(* Logix 5000 project; controller Factory_io vendor 1 type 14 code 15 rev 16.42; software revision 16.03 *)

TASK MainTask (continuous, watchdog 500 ms) : MainProgram

MODULES
   Local : vendor 1 type 14 code 15 (SoftLogixController 2, rev 16.42)
END_MODULES

ADD_ON_INSTRUCTION Add_On_Pusher   (* revision 1.0 *)
VAR_INPUT
   Modo_Op : BOOL; {visible}   // Auto 0 Manual 1
END_VAR
VAR_OUTPUT
   AutoRunning : BOOL;   // Pusher en auto
   ManuRunnig : BOOL;   // Pusher en manual
END_VAR
VAR_INPUT
   cmdRun : BOOL; {visible}   // Activar Pusher Automatico
   cmdStop : BOOL;   // Parada Auto Pusher
END_VAR
VAR_OUTPUT
   StsRunning : BOOL; {visible}   // Salida fisica del PLC
END_VAR
VAR_INPUT
   HMI_Run : BOOL; {visible}   // Pusher Manual
   sensorBackL : BOOL;   // Sensor de posicion del basculante
   sensorFront : BOOL;   // Sensor Posicion basculante
END_VAR
VAR
   HMI_Stop : BOOL;
   expandir : BOOL;
   Encoger : BOOL;   // Accion cuando el sensor Back esta en 0
END_VAR

ROUTINE Logic   (* ladder *)
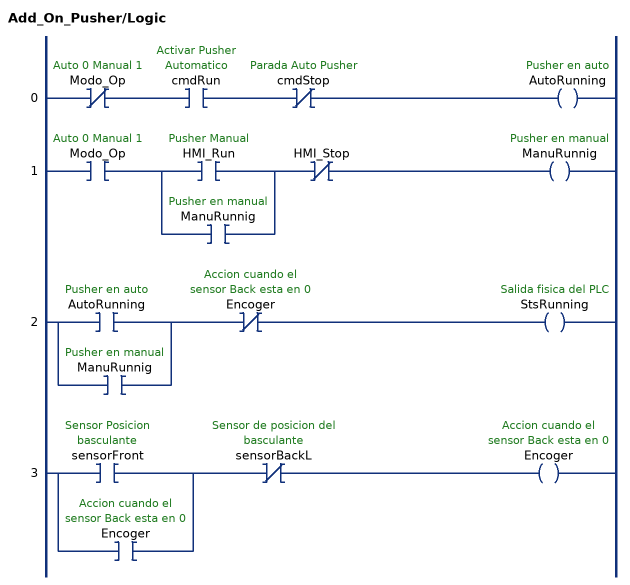
   0: XIO(Modo_Op)XIC(cmdRun)XIO(cmdStop)OTE(AutoRunning);
   1: XIC(Modo_Op)[XIC(HMI_Run) ,XIC(ManuRunnig) ]XIO(HMI_Stop)OTE(ManuRunnig);
   2: [XIC(AutoRunning) ,XIC(ManuRunnig) ]XIO(Encoger)OTE(StsRunning);
   3: [XIC(sensorFront) ,XIC(Encoger) ]XIO(sensorBackL)OTE(Encoger);
END_ROUTINE
END_ADD_ON_INSTRUCTION

ADD_ON_INSTRUCTION Bascula   (* revision 1.0 *)
VAR
   Modo_Op : BOOL;
   HMI_Run : BOOL;
   HMI_Stop : BOOL;
   ManuRunnig : BOOL;
   cmdRun : BOOL;
   cmdStop : BOOL;
   AutoRunning : BOOL;
   Bascula_On : BOOL;
   Peso : REAL;
   Direccion_Derecha : BOOL;
   Ruedas : BOOL;
   Direccion_Izquierda : BOOL;
   Pieza_Izquierda : BOOL;
   Pieza_Derecha : BOOL;
   Sensor_Out_Izquierda : BOOL;
   Sensor_Out_Derecha : BOOL;
END_VAR

ROUTINE Logic   (* ladder *)
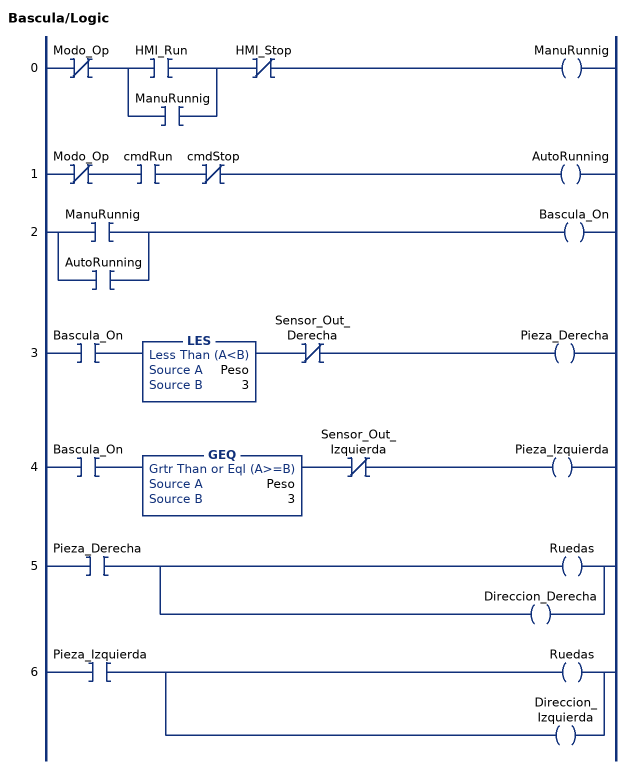
   0: XIO(Modo_Op)[XIC(HMI_Run) ,XIC(ManuRunnig) ]XIO(HMI_Stop)OTE(ManuRunnig);
   1: XIO(Modo_Op)XIC(cmdRun)XIO(cmdStop)OTE(AutoRunning);
   2: [XIC(ManuRunnig) ,XIC(AutoRunning) ]OTE(Bascula_On);
   3: XIC(Bascula_On)LES(Peso,3)XIO(Sensor_Out_Derecha)OTE(Pieza_Derecha);
   4: XIC(Bascula_On)GEQ(Peso,3)XIO(Sensor_Out_Izquierda)OTE(Pieza_Izquierda);
   5: XIC(Pieza_Derecha)[OTE(Ruedas) ,OTE(Direccion_Derecha) ];
   6: XIC(Pieza_Izquierda)[OTE(Ruedas) ,OTE(Direccion_Izquierda) ];
END_ROUTINE
END_ADD_ON_INSTRUCTION

ADD_ON_INSTRUCTION Brazos_Roboticos   (* revision 1.0 *)
VAR_INPUT
   Modo_Op : BOOL; {visible}   // Auto 0 Manual 1
   CmdStop : BOOL; {visible}   // Para desactivar el brazo en modo auto
   CmdRun : BOOL; {visible}   // Para activar el brazo en modo auto
   HMI_Run : BOOL; {visible}   // Para activar el brazo en modo manual
   HMI_Stop : BOOL; {visible}   // Para desactivar el brazo en modo manual
END_VAR
VAR_OUTPUT
   autoRunning : BOOL;   // brazo funcionando en modo auto
   manRunning : BOOL;   // brazo funcionando en modo manual
   StsRunning : BOOL; {visible}   // salida fisica al PLC
END_VAR
VAR_INPUT
   InpRunning : BOOL; {visible}   // Deteccion de falla en el equipo
END_VAR
VAR_OUTPUT
   StsFallo : BOOL; {visible}   // Refleja falla del equipo
   StsStop : BOOL;
END_VAR
VAR
   Timer_TT : BOOL;
   Timer_RES : BOOL;
   Timer_EN : BOOL;
   Timer_DN : BOOL;
   RTO : TIMER;
END_VAR

ROUTINE Logic   (* ladder *)
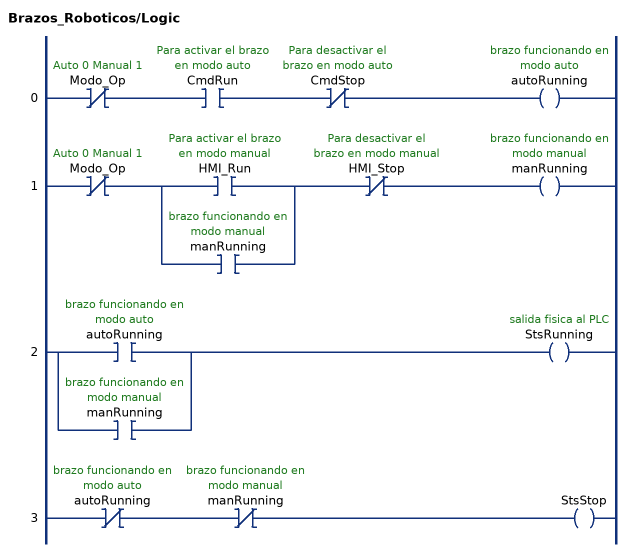
   0: XIO(Modo_Op)XIC(CmdRun)XIO(CmdStop)OTE(autoRunning);
   1: XIO(Modo_Op)[XIC(HMI_Run) ,XIC(manRunning) ]XIO(HMI_Stop)OTE(manRunning);
   2: [XIC(autoRunning) ,XIC(manRunning) ]OTE(StsRunning);
   3: XIO(autoRunning)XIO(manRunning)OTE(StsStop);
END_ROUTINE
END_ADD_ON_INSTRUCTION

ADD_ON_INSTRUCTION Motores   (* revision 1.0 *)
VAR_INPUT
   MODO_OPERACION : BOOL; {visible}
   Cmd_Start : BOOL; {visible}   // Comando para activar el motor en modo auto
   Cmd_Stop : BOOL; {visible}   // Comando para detener el motor en auto
   HMI_Run : BOOL;   // Comando para activar el motor en manual
   HMI_Stop : BOOL;   // Comando para detener el motor en manual
   Inp_Running : BOOL; {visible}   // Confirmacion de arranque del motor
END_VAR
VAR_OUTPUT
   Sts_Running : BOOL; {visible}   // Estado de arranque del motor
   Sts_Running_Pass : BOOL; {visible}   // Estado de motor en la falla
END_VAR
VAR
   Timer_Pass : TIMER := (PRE := 5000);
   Manu_Running : BOOL;
   Auto_Running : BOOL;
END_VAR

ROUTINE Logic   (* ladder *)
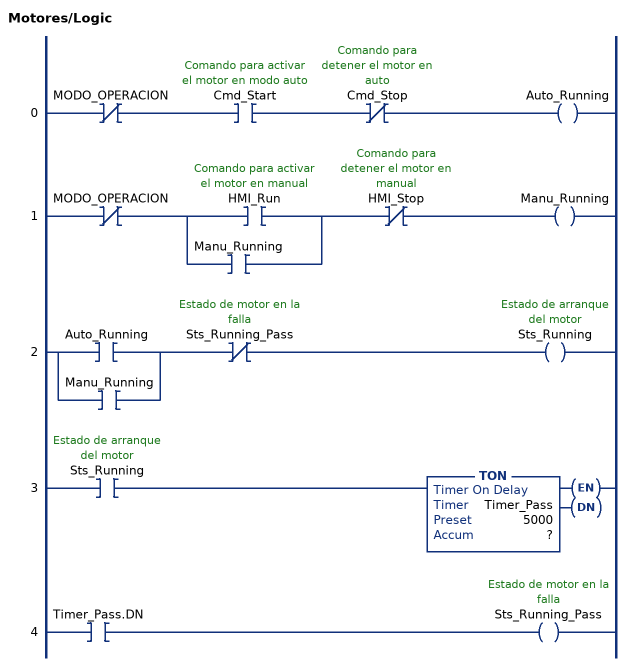
   0: XIO(MODO_OPERACION)XIC(Cmd_Start)XIO(Cmd_Stop)OTE(Auto_Running);
   1: XIO(MODO_OPERACION)[XIC(HMI_Run) ,XIC(Manu_Running) ]XIO(HMI_Stop)OTE(Manu_Running);
   2: [XIC(Auto_Running) ,XIC(Manu_Running) ]XIO(Sts_Running_Pass)OTE(Sts_Running);
   3: XIC(Sts_Running)TON(Timer_Pass,?,?);
   4: XIC(Timer_Pass.DN)OTE(Sts_Running_Pass);
END_ROUTINE
END_ADD_ON_INSTRUCTION

ADD_ON_INSTRUCTION Pick_xyz_avanzado   (* revision 1.0 *)
VAR_INPUT
   Modo_Op : BOOL; {visible}   // Auto 0 Manual 1
END_VAR
VAR_OUTPUT
   AutoRunning : BOOL;   // brazo en auto
   ManuRunnig : BOOL;   // Brazo en manual
END_VAR
VAR_INPUT
   cmdRun : BOOL; {visible}   // Activar Brazo Automatico
   cmdStop : BOOL;   // Parada Auto brazo
END_VAR
VAR_OUTPUT
   StsRunning : BOOL; {visible}   // Salida fisica del PLC
END_VAR
VAR_INPUT
   HMI_Run : BOOL; {visible}   // Brazo Manual
END_VAR
VAR
   HMI_Stop : BOOL;
   maquina_Operando : BOOL;
   Posicion_X : DINT;
   Posicion_Y : DINT;
   Posicion_Z : DINT;
   Etapa_Agarrar : BOOL;
   Etapa_Soltar_1 : BOOL;
   Etapa_Soltar_2 : BOOL;
   Etapa_Soltar_3 : BOOL;
END_VAR

ROUTINE Logic   (* ladder *)
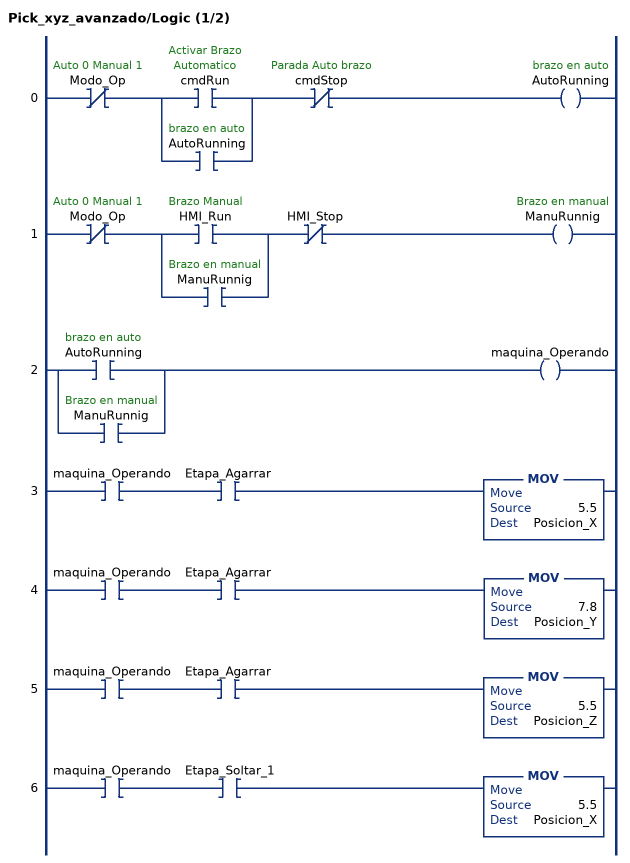
   0: XIO(Modo_Op)[XIC(cmdRun) ,XIC(AutoRunning) ]XIO(cmdStop)OTE(AutoRunning);
   1: XIO(Modo_Op)[XIC(HMI_Run) ,XIC(ManuRunnig) ]XIO(HMI_Stop)OTE(ManuRunnig);
   2: [XIC(AutoRunning) ,XIC(ManuRunnig) ]OTE(maquina_Operando);
   3: XIC(maquina_Operando)XIC(Etapa_Agarrar)MOV(5.5,Posicion_X);
   4: XIC(maquina_Operando)XIC(Etapa_Agarrar)MOV(7.8,Posicion_Y);
   5: XIC(maquina_Operando)XIC(Etapa_Agarrar)MOV(5.5,Posicion_Z);
   6: XIC(maquina_Operando)XIC(Etapa_Soltar_1)MOV(5.5,Posicion_X);
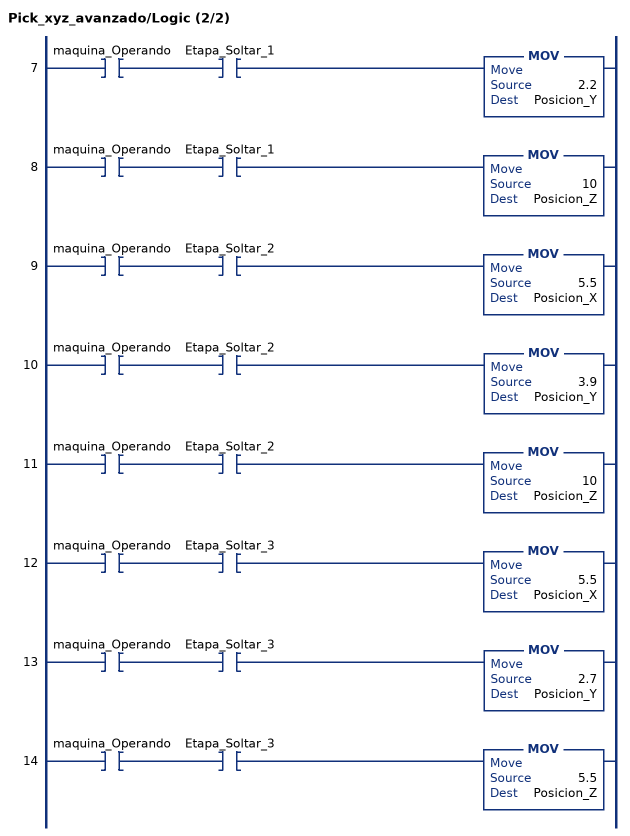
   7: XIC(maquina_Operando)XIC(Etapa_Soltar_1)MOV(2.2,Posicion_Y);
   8: XIC(maquina_Operando)XIC(Etapa_Soltar_1)MOV(10,Posicion_Z);
   9: XIC(maquina_Operando)XIC(Etapa_Soltar_2)MOV(5.5,Posicion_X);
   10: XIC(maquina_Operando)XIC(Etapa_Soltar_2)MOV(3.9,Posicion_Y);
   11: XIC(maquina_Operando)XIC(Etapa_Soltar_2)MOV(10,Posicion_Z);
   12: XIC(maquina_Operando)XIC(Etapa_Soltar_3)MOV(5.5,Posicion_X);
   13: XIC(maquina_Operando)XIC(Etapa_Soltar_3)MOV(2.7,Posicion_Y);
   14: XIC(maquina_Operando)XIC(Etapa_Soltar_3)MOV(5.5,Posicion_Z);
END_ROUTINE
END_ADD_ON_INSTRUCTION

VAR_GLOBAL   (* controller tags *)
   Add_ON_BrazosRoboticos_1 : Brazos_Roboticos;
   Add_ON_BrazosRoboticos_2 : Brazos_Roboticos;
   Add_Pusher_01 : Add_On_Pusher;
   Add_Pusher_02 : Add_On_Pusher;
   Add_Pusher_03 : Add_On_Pusher;
   Agarrar_Soltar : BOOL;
   BOOL_IN_0 : ALIAS FOR Sensor_In1_verde;
   BOOL_IN_1 : ALIAS FOR Sensor_In2_verde;
   BOOL_IN_10 : ALIAS FOR Add_Pusher_03.sensorFront;
   BOOL_IN_11 : ALIAS FOR Add_Pusher_01.sensorBackL;
   BOOL_IN_12 : ALIAS FOR Add_Pusher_02.sensorBackL;
   BOOL_IN_13 : ALIAS FOR Add_Pusher_03.sensorBackL;
   BOOL_IN_14 : ALIAS FOR Difuse_Sensor_In;
   BOOL_IN_15 : ALIAS FOR Difuse_Sensor_Out;
   BOOL_IN_16 : ALIAS FOR Pieza_In;
   BOOL_IN_17 : ALIAS FOR sensor_In_Peso;
   BOOL_IN_18 : ALIAS FOR sensor_Out_banda_der;
   BOOL_IN_19 : ALIAS FOR sensor_Out_banda_Izq;
   BOOL_IN_2 : ALIAS FOR Sensor_Out1;
   BOOL_IN_20 : ALIAS FOR Parada_Peso;
   BOOL_IN_21 : ALIAS FOR Modo_Operacion;
   BOOL_IN_22 : ALIAS FOR STOP;
   BOOL_IN_3 : ALIAS FOR Sensor_Out2;
   BOOL_IN_4 : ALIAS FOR START;
   BOOL_IN_5 : ALIAS FOR sensorVerde;
   BOOL_IN_6 : ALIAS FOR sensorAzul;
   BOOL_IN_7 : ALIAS FOR sensorGris;
   BOOL_IN_8 : ALIAS FOR Add_Pusher_01.sensorFront;
   BOOL_IN_9 : ALIAS FOR Add_Pusher_02.sensorFront;
   BOOL_OUT_0 : ALIAS FOR cintaEntrada1.Sts_Running;
   BOOL_OUT_1 : ALIAS FOR cintaEntrada2.Sts_Running;
   BOOL_OUT_10 : ALIAS FOR cintaEntradaPush2.Sts_Running;
   BOOL_OUT_11 : ALIAS FOR Add_Pusher_01.StsRunning;
   BOOL_OUT_12 : ALIAS FOR Add_Pusher_02.StsRunning;
   BOOL_OUT_13 : ALIAS FOR Add_Pusher_03.StsRunning;
   BOOL_OUT_14 : ALIAS FOR Subir_Bajar;
   BOOL_OUT_15 : ALIAS FOR Agarrar_Soltar;
   BOOL_OUT_16 : ALIAS FOR Pasa_Banda;
   BOOL_OUT_17 : ALIAS FOR Cinta_In_Pick1.Sts_Running;
   BOOL_OUT_18 : ALIAS FOR Cinta_In_Pick2.Sts_Running;
   BOOL_OUT_19 : ALIAS FOR Cinta_In_Pick3.Sts_Running;
   BOOL_OUT_2 : ALIAS FOR cintaSalida_01.Sts_Running;
   BOOL_OUT_20 : ALIAS FOR Cinta_In_Pick4.Sts_Running;
   BOOL_OUT_21 : ALIAS FOR Cinta_In_Pick5.Sts_Running;
   BOOL_OUT_22 : ALIAS FOR Cinta_In_Pick6.Sts_Running;
   BOOL_OUT_23 : ALIAS FOR cintaPP.Sts_Running;
   BOOL_OUT_24 : ALIAS FOR movScale.Sts_Running;
   BOOL_OUT_25 : ALIAS FOR clasificaPlus.Sts_Running;
   BOOL_OUT_26 : ALIAS FOR clasificaDerecha.Sts_Running;
   BOOL_OUT_27 : ALIAS FOR clasificaIzq.Sts_Running;
   BOOL_OUT_28 : ALIAS FOR cintaPesoDer.Sts_Running;
   BOOL_OUT_29 : ALIAS FOR cintaPesoIzq.Sts_Running;
   BOOL_OUT_3 : ALIAS FOR cintaSalida_02.Sts_Running;
   BOOL_OUT_30 : ALIAS FOR Luz_Verde;
   BOOL_OUT_31 : ALIAS FOR Luz_stop;
   BOOL_OUT_4 : ALIAS FOR Maquina_1;
   BOOL_OUT_5 : ALIAS FOR Maquina_2;
   BOOL_OUT_6 : ALIAS FOR cintaRecorrido1.Sts_Running;
   BOOL_OUT_7 : ALIAS FOR cintaRecorrido2.Sts_Running;
   BOOL_OUT_8 : ALIAS FOR cintarecorrido3.Sts_Running;
   BOOL_OUT_9 : ALIAS FOR cintaEntradaPush1.Sts_Running;
   cinta : Motores;
   Cinta_In_Pick1 : Motores;
   Cinta_In_Pick2 : Motores;
   Cinta_In_Pick3 : Motores;
   Cinta_In_Pick4 : Motores;
   Cinta_In_Pick5 : Motores;
   Cinta_In_Pick6 : Motores;
   cintaEntrada1 : Motores;
   cintaEntrada1_01 : Motores;
   cintaEntrada1_02 : Motores;
   cintaEntrada2 : Motores;
   cintaEntradaPush1 : Motores;
   cintaEntradaPush2 : Motores;
   cintaPeso : Motores;
   cintaPesoDer : Motores;
   cintaPesoIzq : Motores;
   cintaPP : Motores;
   cintaRecorrido1 : Motores;
   cintaRecorrido2 : Motores;
   cintarecorrido3 : Motores;
   cintarecorrido3_01 : Motores;
   cintaSalida_01 : Motores;
   cintaSalida_02 : Motores;
   cintaSalida_03 : Motores;
   cintaSalida_04 : Motores;
   cintaSalida_05 : Motores;
   cintaSalida_06 : Motores;
   clasificaDerecha : Motores;
   clasificaIzq : Motores;
   clasificaPlus : Motores;
   Difuse_Sensor_In : BOOL;
   Difuse_Sensor_Out : BOOL;
   FLOAT_IN_0 : ALIAS FOR SensorPeso;
   INICO_001 : SFC_STEP := (Status := 16#0800_0201, DN := 1, T := 16, TMax := 20306, Count := 4);
   INICO_002 : SFC_STEP := (Status := 16#0800_0201, DN := 1, T := 16, TMax := 20306, Count := 4);
   Luz_stop : BOOL;
   Luz_Verde : BOOL;
   Maquina_1 : BOOL;
   Maquina_2 : BOOL;
   Modo_Operacion : BOOL;   // 0 AUTO 1 MANUAL
   movScale : Motores;
   Parada_Peso : BOOL;
   Pasa_Banda : BOOL;
   Pick_On : BOOL;
   Pieza_In : BOOL;
   Sensor_In1_verde : BOOL := 1;
   Sensor_In2_verde : BOOL := 1;
   sensor_In_Peso : BOOL;
   Sensor_Out1 : BOOL := 1;
   Sensor_Out2 : BOOL := 1;
   sensor_Out_banda_der : BOOL;
   sensor_Out_banda_Izq : BOOL;
   sensorAzul : BOOL;
   sensorGris : BOOL;
   SensorPeso : REAL;
   sensorVerde : BOOL;
   START : BOOL;
   STOP : BOOL;
   Subir_Bajar : BOOL;
   SYS_ON : BOOL;
END_VAR

PROGRAM MainProgram   (* main routine MainRoutine *)
VAR
   Action_000 : SFC_ACTION := (Status := 16#c000_0000, A := 1, Q := 1, Count := 4);
   Action_001 : SFC_ACTION := (Count := 4);
   Action_002 : SFC_ACTION := (Count := 4);
   Action_003 : SFC_ACTION := (Count := 3);
   Action_004 : SFC_ACTION := (Count := 4);
   Action_005 : SFC_ACTION := (Status := 16#c000_0000, A := 1, Q := 1, Count := 4);
   Action_006 : SFC_ACTION := (Count := 3);
   Action_007 : SFC_ACTION := (Count := 4);
   Action_008 : SFC_ACTION;
   Action_009 : SFC_ACTION;
   Action_010 : SFC_ACTION;
   Action_011 : SFC_ACTION;
   Action_012 : SFC_ACTION;
   Action_013 : SFC_ACTION;
   Action_014 : SFC_ACTION;
   Action_015 : SFC_ACTION;
   Action_016 : SFC_ACTION;
   Action_017 : SFC_ACTION;
   Action_018 : SFC_ACTION;
   Action_019 : SFC_ACTION;
   Motores_01 : Motores := (Cmd_Start := 1);
   Motores_02 : Motores := (Cmd_Start := 1);
   Motores_03 : Motores := (Cmd_Start := 1);
   Motores_04 : Motores := (Cmd_Start := 1);
   Step_000 : SFC_STEP;
   Step_001 : SFC_STEP;
   Step_002 : SFC_STEP := (Status := 16#0800_0001, DN := 1, PRE := 400, T := 314, TMax := 327, Count := 4);
   Step_003 : SFC_STEP := (Status := 16#0800_0001, DN := 1, T := 2150, TMax := 2212, Count := 4);
   Step_004 : SFC_STEP := (Status := 16#0800_0001, DN := 1, T := 2192, TMax := 2234, Count := 4);
   Step_005 : SFC_STEP := (PRE := 300);
   Step_006 : SFC_STEP := (Status := 16#0800_0001, DN := 1, T := 18, TMax := 19, Count := 4);
   Step_007 : SFC_STEP := (Status := 16#0800_0001, DN := 1, T := 18, TMax := 19, Count := 4);
   Step_008 : SFC_STEP := (Status := 16#a800_0001, X := 1, SA := 1, DN := 1, T := 60168, TMax := 60168, Count := 4);
   Step_009 : SFC_STEP := (Status := 16#0800_0001, DN := 1, PRE := 6000, T := 5019, TMax := 5019, Count := 3);
   Step_010 : SFC_STEP := (Status := 16#a800_0001, X := 1, SA := 1, DN := 1, T := 60169, TMax := 60169, Count := 4);
   Step_011 : SFC_STEP := (Status := 16#0800_0001, DN := 1, PRE := 400, T := 314, TMax := 322, Count := 4);
   Step_012 : SFC_STEP := (Status := 16#0800_0001, DN := 1, PRE := 2000, T := 5019, TMax := 5019, Count := 3);
   Step_013 : SFC_STEP;
   Step_014 : SFC_STEP;
   Step_015 : SFC_STEP := (PRE := 300);
   Step_016 : SFC_STEP := (PRE := 400);
   Step_017 : SFC_STEP := (PRE := 400);
   Step_018 : SFC_STEP := (PRE := 1000);
   Step_019 : SFC_STEP;
   Step_020 : SFC_STEP := (PRE := 300);
   Step_021 : SFC_STEP := (PRE := 500);
   Step_022 : SFC_STEP := (PRE := 300);
   Step_023 : SFC_STEP;
   Step_024 : SFC_STEP;
   Step_025 : SFC_STEP := (PRE := 3100);
   Step_026 : SFC_STEP := (PRE := 3100);
   Step_027 : SFC_STEP;
   Step_028 : SFC_STEP := (PRE := 200);
   Tran_000 : BOOL;
   Tran_001 : BOOL := 1;
   Tran_002 : BOOL := 1;
   Tran_003 : BOOL := 1;
   Tran_004 : BOOL := 1;
   Tran_005 : BOOL := 1;
   Tran_006 : BOOL;
   Tran_007 : BOOL := 1;
   Tran_008 : BOOL := 1;
   Tran_009 : BOOL := 1;
   Tran_010 : BOOL := 1;
   Tran_011 : BOOL;
   Tran_012 : BOOL := 1;
   Tran_013 : BOOL;
   Tran_014 : BOOL;
   Tran_015 : BOOL;
   Tran_016 : BOOL;
   Tran_017 : BOOL;
   Tran_018 : BOOL;
   Tran_019 : BOOL;
   Tran_020 : BOOL;
   Tran_021 : BOOL;
   Tran_022 : BOOL;
   Tran_023 : BOOL;
   Tran_024 : BOOL;
   Tran_025 : BOOL;
   Tran_026 : BOOL;
   Tran_027 : BOOL;
   Tran_028 : BOOL;
END_VAR

ROUTINE BRAZOS_ROBOTICOS   (* sequential function chart *)
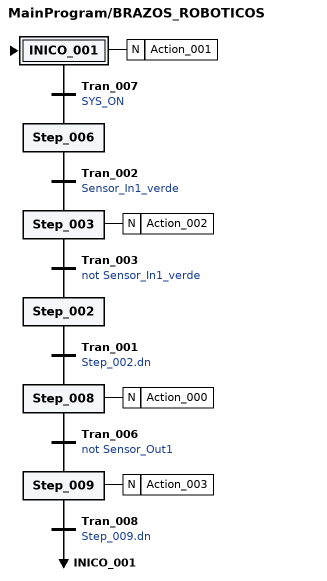
   INITIAL_STEP INICO_001:
      ACTION Action_001 (N):
         cintaEntrada1.Cmd_Start:=0;
         cintaSalida_01.Cmd_Start:=0;
         Maquina_1:=0;
         
         
         
      END_ACTION
   END_STEP
   TRANSITION Tran_007 FROM INICO_001 TO Step_006
      := SYS_ON
   END_TRANSITION
   STEP Step_006:
   END_STEP
   TRANSITION Tran_002 FROM Step_006 TO Step_003
      :=  Sensor_In1_verde
   END_TRANSITION
   STEP Step_003:
      ACTION Action_002 (N):
         cintaEntrada1.Cmd_Start:=1;
         
      END_ACTION
   END_STEP
   TRANSITION Tran_003 FROM Step_003 TO Step_002
      := not Sensor_In1_verde
   END_TRANSITION
   STEP Step_002:
   END_STEP
   TRANSITION Tran_001 FROM Step_002 TO Step_008
      := Step_002.dn
   END_TRANSITION
   STEP Step_008:
      ACTION Action_000 (N):
         cintaEntrada1.Cmd_Start:=0;
         Maquina_1:=1;
      END_ACTION
   END_STEP
   TRANSITION Tran_006 FROM Step_008 TO Step_009
      := not Sensor_Out1
   END_TRANSITION
   STEP Step_009:
      ACTION Action_003 (N):
         cintaSalida_01.Cmd_Start:=1;
         
         
      END_ACTION
   END_STEP
   TRANSITION Tran_008 FROM Step_009 TO INICO_001
      := Step_009.dn
   END_TRANSITION
END_ROUTINE

ROUTINE BRAZOS_ROBOTICOS_TAPAS   (* sequential function chart *)
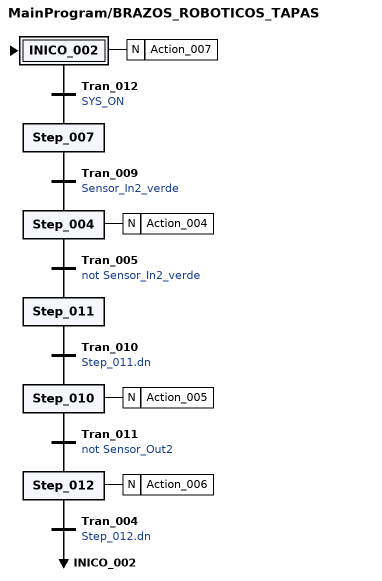
   INITIAL_STEP INICO_002:
      ACTION Action_007 (N):
         cintaEntrada2.Cmd_Start:=0;
         cintaSalida_02.Cmd_Start:=0;
         Maquina_2:=0;
         
         
         
      END_ACTION
   END_STEP
   TRANSITION Tran_012 FROM INICO_002 TO Step_007
      := SYS_ON
   END_TRANSITION
   STEP Step_007:
   END_STEP
   TRANSITION Tran_009 FROM Step_007 TO Step_004
      :=  Sensor_In2_verde
   END_TRANSITION
   STEP Step_004:
      ACTION Action_004 (N):
         cintaEntrada2.Cmd_Start:=1;
         
      END_ACTION
   END_STEP
   TRANSITION Tran_005 FROM Step_004 TO Step_011
      := not Sensor_In2_verde
   END_TRANSITION
   STEP Step_011:
   END_STEP
   TRANSITION Tran_010 FROM Step_011 TO Step_010
      := Step_011.dn
   END_TRANSITION
   STEP Step_010:
      ACTION Action_005 (N):
         cintaEntrada2.Cmd_Start:=0;
         Maquina_2:=1;
      END_ACTION
   END_STEP
   TRANSITION Tran_011 FROM Step_010 TO Step_012
      := not Sensor_Out2
   END_TRANSITION
   STEP Step_012:
      ACTION Action_006 (N):
         cintaSalida_02.Cmd_Start:=1;
         cintarecorrido3.Cmd_Start:=1;
         
         
      END_ACTION
   END_STEP
   TRANSITION Tran_004 FROM Step_012 TO INICO_002
      := Step_012.dn
   END_TRANSITION
END_ROUTINE

ROUTINE cintas_pushers   (* function block diagram *)
   SHEET 1
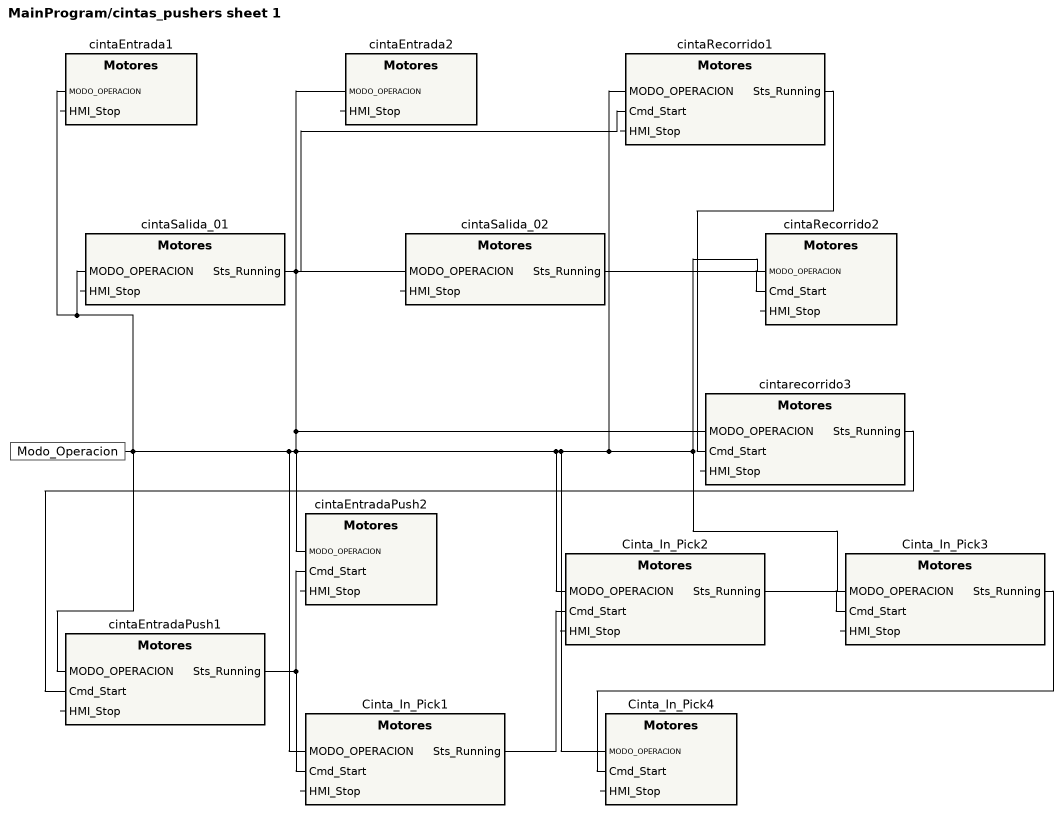
   cintaEntrada1 : Motores(MODO_OPERACION := Modo_Operacion);   // unwired pins: HMI_Stop
   cintaSalida_01 : Motores(MODO_OPERACION := Modo_Operacion);   // unwired pins: HMI_Stop
   cintaEntrada2 : Motores(MODO_OPERACION := Modo_Operacion);   // unwired pins: HMI_Stop
   cintaSalida_02 : Motores(MODO_OPERACION := Modo_Operacion);   // unwired pins: HMI_Stop
   cintaRecorrido1 : Motores(MODO_OPERACION := Modo_Operacion, Cmd_Start := cintaSalida_01.Sts_Running);   // unwired pins: HMI_Stop
   cintarecorrido3 : Motores(MODO_OPERACION := Modo_Operacion, Cmd_Start := cintaRecorrido1.Sts_Running);   // unwired pins: HMI_Stop
   cintaEntradaPush1 : Motores(MODO_OPERACION := Modo_Operacion, Cmd_Start := cintarecorrido3.Sts_Running);   // unwired pins: HMI_Stop
   cintaEntradaPush2 : Motores(MODO_OPERACION := Modo_Operacion, Cmd_Start := cintaEntradaPush1.Sts_Running);   // unwired pins: HMI_Stop
   Cinta_In_Pick1 : Motores(MODO_OPERACION := Modo_Operacion, Cmd_Start := cintaEntradaPush1.Sts_Running);   // unwired pins: HMI_Stop
   Cinta_In_Pick2 : Motores(MODO_OPERACION := Modo_Operacion, Cmd_Start := Cinta_In_Pick1.Sts_Running);   // unwired pins: HMI_Stop
   cintaRecorrido2 : Motores(MODO_OPERACION := Modo_Operacion, Cmd_Start := cintaSalida_02.Sts_Running);   // unwired pins: HMI_Stop
   Cinta_In_Pick3 : Motores(MODO_OPERACION := Modo_Operacion, Cmd_Start := Cinta_In_Pick2.Sts_Running);   // unwired pins: HMI_Stop
   Cinta_In_Pick4 : Motores(MODO_OPERACION := Modo_Operacion, Cmd_Start := Cinta_In_Pick3.Sts_Running);   // unwired pins: HMI_Stop
   SHEET 2
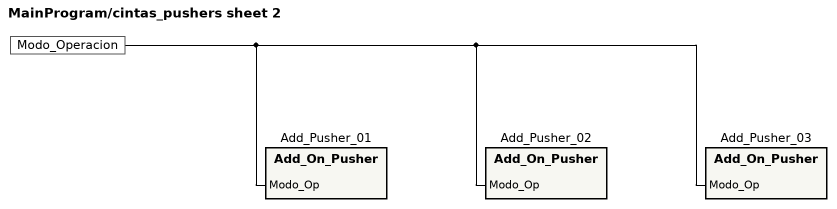
   Add_Pusher_01 : Add_On_Pusher(Modo_Op := Modo_Operacion);
   Add_Pusher_02 : Add_On_Pusher(Modo_Op := Modo_Operacion);
   Add_Pusher_03 : Add_On_Pusher(Modo_Op := Modo_Operacion);
   SHEET 3
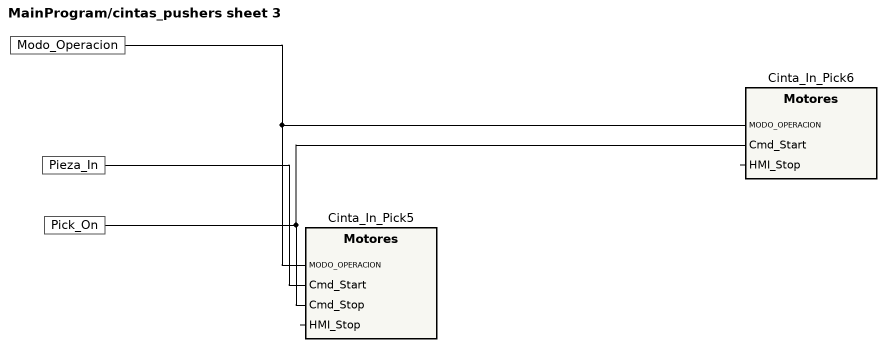
   Cinta_In_Pick5 : Motores(MODO_OPERACION := Modo_Operacion, Cmd_Start := Pieza_In, Cmd_Stop := Pick_On);   // unwired pins: HMI_Stop
   Cinta_In_Pick6 : Motores(MODO_OPERACION := Modo_Operacion, Cmd_Start := Pick_On);   // unwired pins: HMI_Stop
   SHEET 4
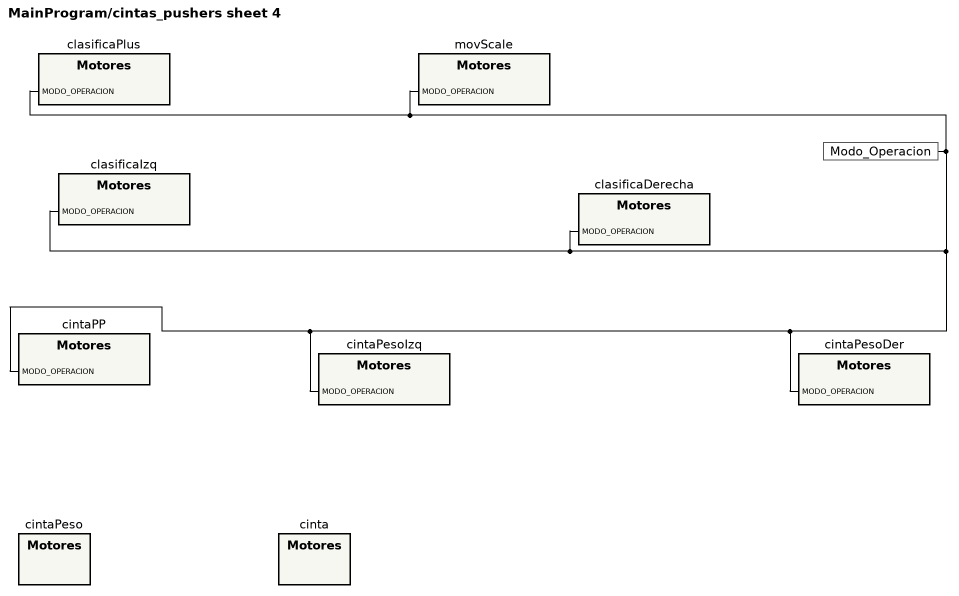
   cintaPeso : Motores();
   cinta : Motores();
   cintaPP : Motores(MODO_OPERACION := Modo_Operacion);
   clasificaPlus : Motores(MODO_OPERACION := Modo_Operacion);
   clasificaIzq : Motores(MODO_OPERACION := Modo_Operacion);
   cintaPesoIzq : Motores(MODO_OPERACION := Modo_Operacion);
   movScale : Motores(MODO_OPERACION := Modo_Operacion);
   clasificaDerecha : Motores(MODO_OPERACION := Modo_Operacion);
   cintaPesoDer : Motores(MODO_OPERACION := Modo_Operacion);
END_ROUTINE

ROUTINE Distribucion_por_peso   (* sequential function chart *)
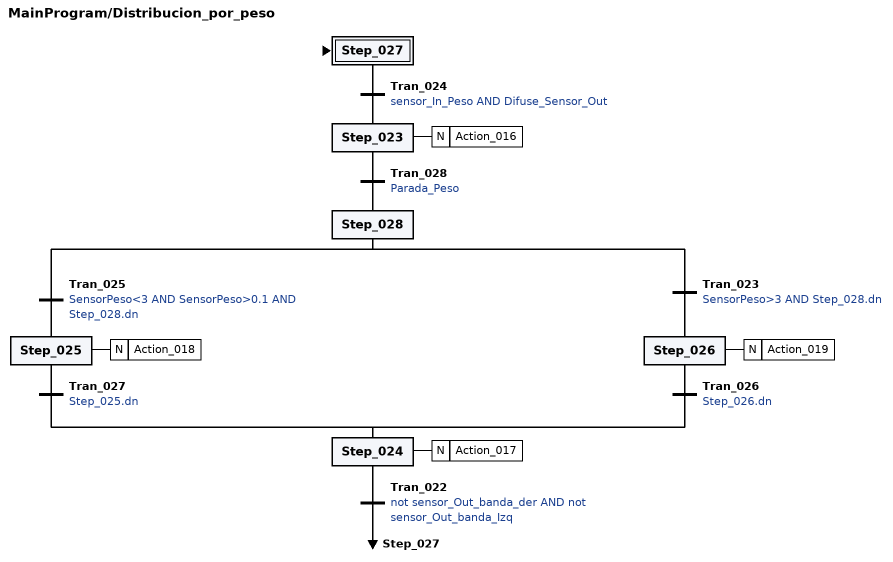
   INITIAL_STEP Step_027:
   END_STEP
   TRANSITION Tran_024 FROM Step_027 TO Step_023
      := sensor_In_Peso AND Difuse_Sensor_Out
   END_TRANSITION
   STEP Step_023:
      ACTION Action_016 (N):
         movScale.Sts_Running:=1;
         cintaPP.Sts_Running:=1;
      END_ACTION
   END_STEP
   TRANSITION Tran_028 FROM Step_023 TO Step_028
      := Parada_Peso
   END_TRANSITION
   STEP Step_028:
   END_STEP
   TRANSITION Tran_025 FROM Step_028 TO Step_025
      := SensorPeso<3 AND SensorPeso>0.1 AND Step_028.dn
   END_TRANSITION
   TRANSITION Tran_023 FROM Step_028 TO Step_026
      := SensorPeso>3 AND Step_028.dn
   END_TRANSITION
   STEP Step_025:
      ACTION Action_018 (N):
         clasificaPlus.Sts_Running:=1;
         clasificaDerecha.Sts_Running:=1;
         cintaPesoDer.Sts_Running:=1;
         movScale.Sts_Running:=1;
      END_ACTION
   END_STEP
   STEP Step_026:
      ACTION Action_019 (N):
         clasificaPlus.Sts_Running:=1;
         clasificaIzq.Sts_Running:=1;
         cintaPesoIzq.Sts_Running:=1;
         movScale.Sts_Running:=1;
      END_ACTION
   END_STEP
   TRANSITION Tran_026 FROM Step_026 TO Step_024
      :=  Step_026.dn
   END_TRANSITION
   TRANSITION Tran_027 FROM Step_025 TO Step_024
      :=  Step_025.dn
   END_TRANSITION
   STEP Step_024:
      ACTION Action_017 (N):
         clasificaPlus.Sts_Running:=0;
         clasificaDerecha.Sts_Running:=0;
         cintaPesoDer.Sts_Running:=0;
         clasificaIzq.Sts_Running:=0;
         cintaPesoIzq.Sts_Running:=0;
      END_ACTION
   END_STEP
   TRANSITION Tran_022 FROM Step_024 TO Step_027
      := not sensor_Out_banda_der AND not sensor_Out_banda_Izq
   END_TRANSITION
END_ROUTINE

ROUTINE MainRoutine   (* ladder *)
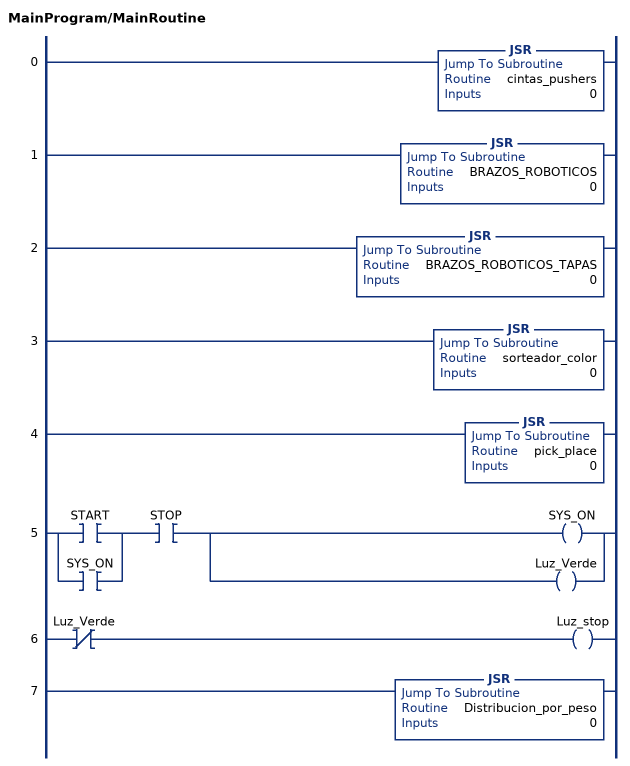
   0: JSR(cintas_pushers,0);
   1: JSR(BRAZOS_ROBOTICOS,0);
   2: JSR(BRAZOS_ROBOTICOS_TAPAS,0);
   3: JSR(sorteador_color,0);
   4: JSR(pick_place,0);
   5: [XIC(START) ,XIC(SYS_ON) ]XIC(STOP)[OTE(SYS_ON) ,OTE(Luz_Verde) ];
   6: XIO(Luz_Verde)OTE(Luz_stop);
   7: JSR(Distribucion_por_peso,0);
END_ROUTINE

ROUTINE pick_place   (* sequential function chart *)
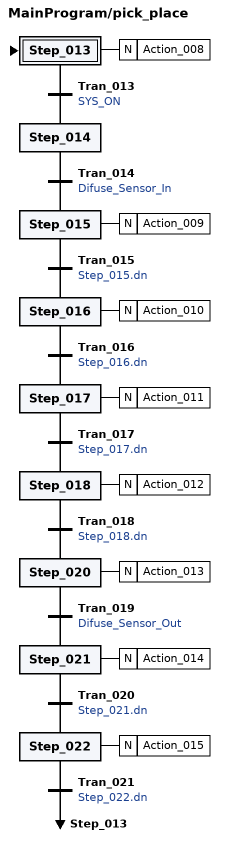
   INITIAL_STEP Step_013:
      ACTION Action_008 (N):
         Subir_Bajar:=0;
         Agarrar_Soltar:=0;
         Pasa_Banda:=0;
         Pick_On:=0;
      END_ACTION
   END_STEP
   TRANSITION Tran_013 FROM Step_013 TO Step_014
      := SYS_ON
   END_TRANSITION
   STEP Step_014:
   END_STEP
   TRANSITION Tran_014 FROM Step_014 TO Step_015
      := Difuse_Sensor_In
   END_TRANSITION
   STEP Step_015:
      ACTION Action_009 (N):
         Subir_Bajar:=1;
         Pick_On:=1;
      END_ACTION
   END_STEP
   TRANSITION Tran_015 FROM Step_015 TO Step_016
      := Step_015.dn
   END_TRANSITION
   STEP Step_016:
      ACTION Action_010 (N):
         Agarrar_Soltar:=1;
         Subir_Bajar:=1;
         Pick_On:=1;
      END_ACTION
   END_STEP
   TRANSITION Tran_016 FROM Step_016 TO Step_017
      := Step_016.dn
   END_TRANSITION
   STEP Step_017:
      ACTION Action_011 (N):
         Subir_Bajar:=0;
         Agarrar_Soltar:=1;
         Pick_On:=1;
      END_ACTION
   END_STEP
   TRANSITION Tran_017 FROM Step_017 TO Step_018
      := Step_017.dn
   END_TRANSITION
   STEP Step_018:
      ACTION Action_012 (N):
         Pasa_Banda:=1;
         Agarrar_Soltar:=1;
         Pick_On:=1;
      END_ACTION
   END_STEP
   TRANSITION Tran_018 FROM Step_018 TO Step_020
      := Step_018.dn
   END_TRANSITION
   STEP Step_020:
      ACTION Action_013 (N):
         Subir_Bajar:=1;
         Agarrar_Soltar:=1;
         Pick_On:=1;
         
      END_ACTION
   END_STEP
   TRANSITION Tran_019 FROM Step_020 TO Step_021
      := Difuse_Sensor_Out
   END_TRANSITION
   STEP Step_021:
      ACTION Action_014 (N):
         Agarrar_Soltar:=0;
         Pick_On:=1;
         
      END_ACTION
   END_STEP
   TRANSITION Tran_020 FROM Step_021 TO Step_022
      := Step_021.dn
   END_TRANSITION
   STEP Step_022:
      ACTION Action_015 (N):
         Subir_Bajar:=0;
         Pick_On:=1;
      END_ACTION
   END_STEP
   TRANSITION Tran_021 FROM Step_022 TO Step_013
      := Step_022.dn
   END_TRANSITION
END_ROUTINE

ROUTINE sorteador_color   (* ladder *)
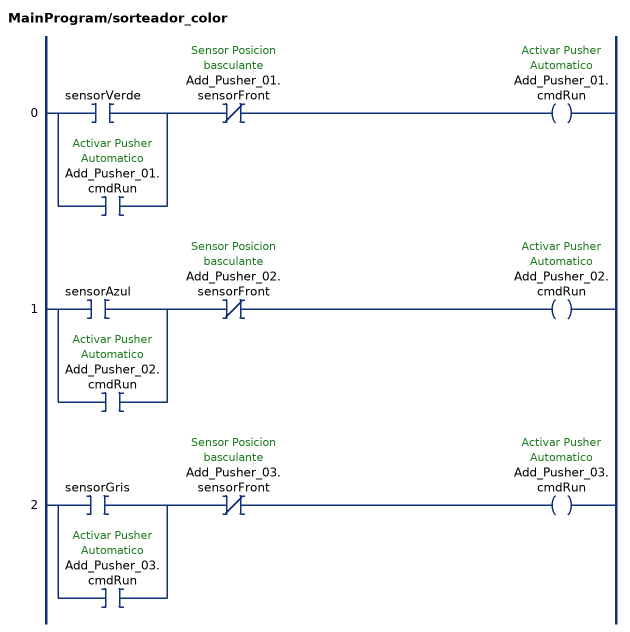
   0: [XIC(sensorVerde) ,XIC(Add_Pusher_01.cmdRun) ]XIO(Add_Pusher_01.sensorFront)OTE(Add_Pusher_01.cmdRun);
   1: [XIC(sensorAzul) ,XIC(Add_Pusher_02.cmdRun) ]XIO(Add_Pusher_02.sensorFront)OTE(Add_Pusher_02.cmdRun);
   2: [XIC(sensorGris) ,XIC(Add_Pusher_03.cmdRun) ]XIO(Add_Pusher_03.sensorFront)OTE(Add_Pusher_03.cmdRun);
END_ROUTINE
END_PROGRAM
